// TIA Portal V20 export
// export: Created 2025-12-01T14:57:00.0403438Z, ExportSetting None, DisplayName Totally Integrated Automation Portal, DisplayVersion V20 Update 3, DisplayName TIA Portal Openness, DisplayVersion V20 Update 3, DisplayName TIA Portal Version Control Interface, DisplayVersion V20 Update 3, DisplayName STEP 7 Professional, DisplayVersion V20 Update 3, DisplayName STEP 7 Safety, DisplayVersion V20 Update 2, DisplayName WinCC Basic/Comfort/Advanced, DisplayVersion V20 Update 3, DisplayName WinCC Professional, DisplayVersion V20 Update 3, DisplayName WinCC Unified, DisplayVersion V20 Update 3
FUNCTION "FC427_TL_Sep_Salida_Bidi" : Void   // FC427, LAD
{ S7_Optimized_Access := 'FALSE' }
AUTHOR : TLigero
NAME : 20160208
VERSION : 3.1
// FECHA:    27/07/2014  AUTOR: G.Martin
// INSTALACION: Magyar Posta
// //////////////////////////////////
// // Registro Incidencias   ////////
// //////////////////////////////////
// FECHA:21/10/14   AUTOR MODIFICACION: N.Rodriguez
// DESCRIPCION: 
// Adaptación de la función al estandar actual
// 
// FECHA:   AUTOR MODIFICACION: 
// DESCRIPCION:
// stored: AutoNumber false, SetENOAutomatically false
   VAR_INPUT
      Mesa : UInt;
      En_Tension : Bool;
      Phs_Tx_E1 : Bool;   // Se utiliza esta fotocelula en caga E1-E3
      Phs_Tx_E3 : Bool;   // Se utiliza esta fotocelula en caga E3-E1
      Termico_Tx : Bool;
      Avance_E1_Tx_Ok : Bool;   // Avance con dirección E1-E3
      Avance_E3_Tx_Ok : Bool;   // Avance con dirección E3-E1
      Modo_Pasoapaso_Tx : Bool;
      Direccion_Inv_Tx : Bool;
      AVTF_Ent_M1 : Bool;
      AVTF_Ent_M3 : Bool;
      PTF_Sal_M1 : Bool;
      NXT_Avance_M1 : Bool;
      PTF_Sal_M3 : Bool;
      NXT_Avance_M3 : Bool;
      V_Ausencia_Tms : UDInt;
      V_Paro : UDInt;
      V_Separacion : UDInt;
      V_Caja_Max : UDInt;
      V_TOut_Tx_Mx : UDInt;
      V_Acumulacion : UDInt;
      V_Ausencia : UDInt;
   END_VAR
   VAR_OUTPUT
      PTF_Ent_M1 : Bool;
      PTF_Ent_M3 : Bool;
      AVTF_Sal_M1 : Bool;
      AVTF_Sal_M3 : Bool;
   END_VAR
   VAR_IN_OUT
      NXT_Descarga_Act_M1 : Bool;
      NXT_Descarga_Act_M3 : Bool;
      Carga_Activa_Tx : Bool;
      Carga_Activa_Inv_TX : Bool;
      MAUX_FN_Avtf : Bool;
      MAUX_FN_Direc : Bool;
      MAUX_FP_Direc : Bool;
      Mem_CNT_Tmp_AUS : Bool;
      Mem_CNT_Tmp_Paro_Tx : Bool;
      Mem_CNT_Acumulacion : Bool;
   END_VAR
   VAR_TEMP
      CNT_Sep : Word;
      CNT_Sep_FORZ_Sep : Int;
      Aux_Parar : Bool;
      Mem_CNT_Separacion : Bool;
      mem_atasco : Bool;
      fp_direc : Bool;
      fn_direc : Bool;
      mem_atasco_inv : Bool;
      ok_tension : Bool;
   END_VAR
   VAR_TEMP   // added for the SCL form of the ladder/FBD networks
      _w1 : Bool;
      _w2 : Bool;
   END_VAR
BEGIN

REGION Network 1: Marca General Error
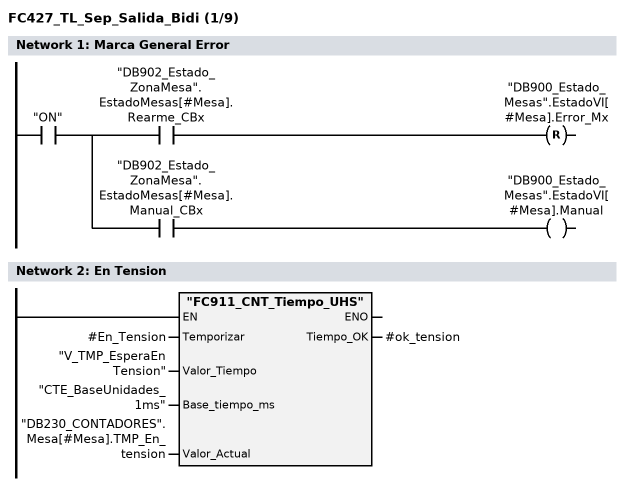
   RUNG wire#powerrail
      Contact( "ON" )
      wire#w1
      Contact( "DB902_Estado_ZonaMesa".EstadoMesas[#Mesa].Rearme_CBx )
      R_Coil( "DB900_Estado_Mesas".EstadoVI[#Mesa].Error_Mx )
   END_RUNG
   RUNG wire#w1
      Contact( "DB902_Estado_ZonaMesa".EstadoMesas[#Mesa].Manual_CBx )
      Coil( "DB900_Estado_Mesas".EstadoVI[#Mesa].Manual )
   END_RUNG
   // the same network as SCL:
   IF "ON" AND "DB902_Estado_ZonaMesa".EstadoMesas[#Mesa].Rearme_CBx THEN
       "DB900_Estado_Mesas".EstadoVI[#Mesa].Error_Mx := FALSE;
   END_IF;
   "DB900_Estado_Mesas".EstadoVI[#Mesa].Manual := "ON" AND "DB902_Estado_ZonaMesa".EstadoMesas[#Mesa].Manual_CBx;
END_REGION

REGION Network 2: En Tension
   RUNG wire#powerrail
      "FC911_CNT_Tiempo_UHS"(Temporizar := #En_Tension, Valor_Tiempo := "V_TMP_EsperaEnTension", Base_tiempo_ms := "CTE_BaseUnidades_1ms", Valor_Actual := "DB230_CONTADORES".Mesa[#Mesa].TMP_En_tension, Tiempo_OK => #ok_tension)
   END_RUNG
   // the same network as SCL:
   "FC911_CNT_Tiempo_UHS"(Temporizar := #En_Tension,
                          Valor_Tiempo := "V_TMP_EsperaEnTension",
                          Base_tiempo_ms := "CTE_BaseUnidades_1ms",
                          Valor_Actual := "DB230_CONTADORES".Mesa[#Mesa].TMP_En_tension,
                          Tiempo_OK => #ok_tension);
END_REGION

REGION Network 3: Reseteamos las marcas cuando hay cambio de direccion
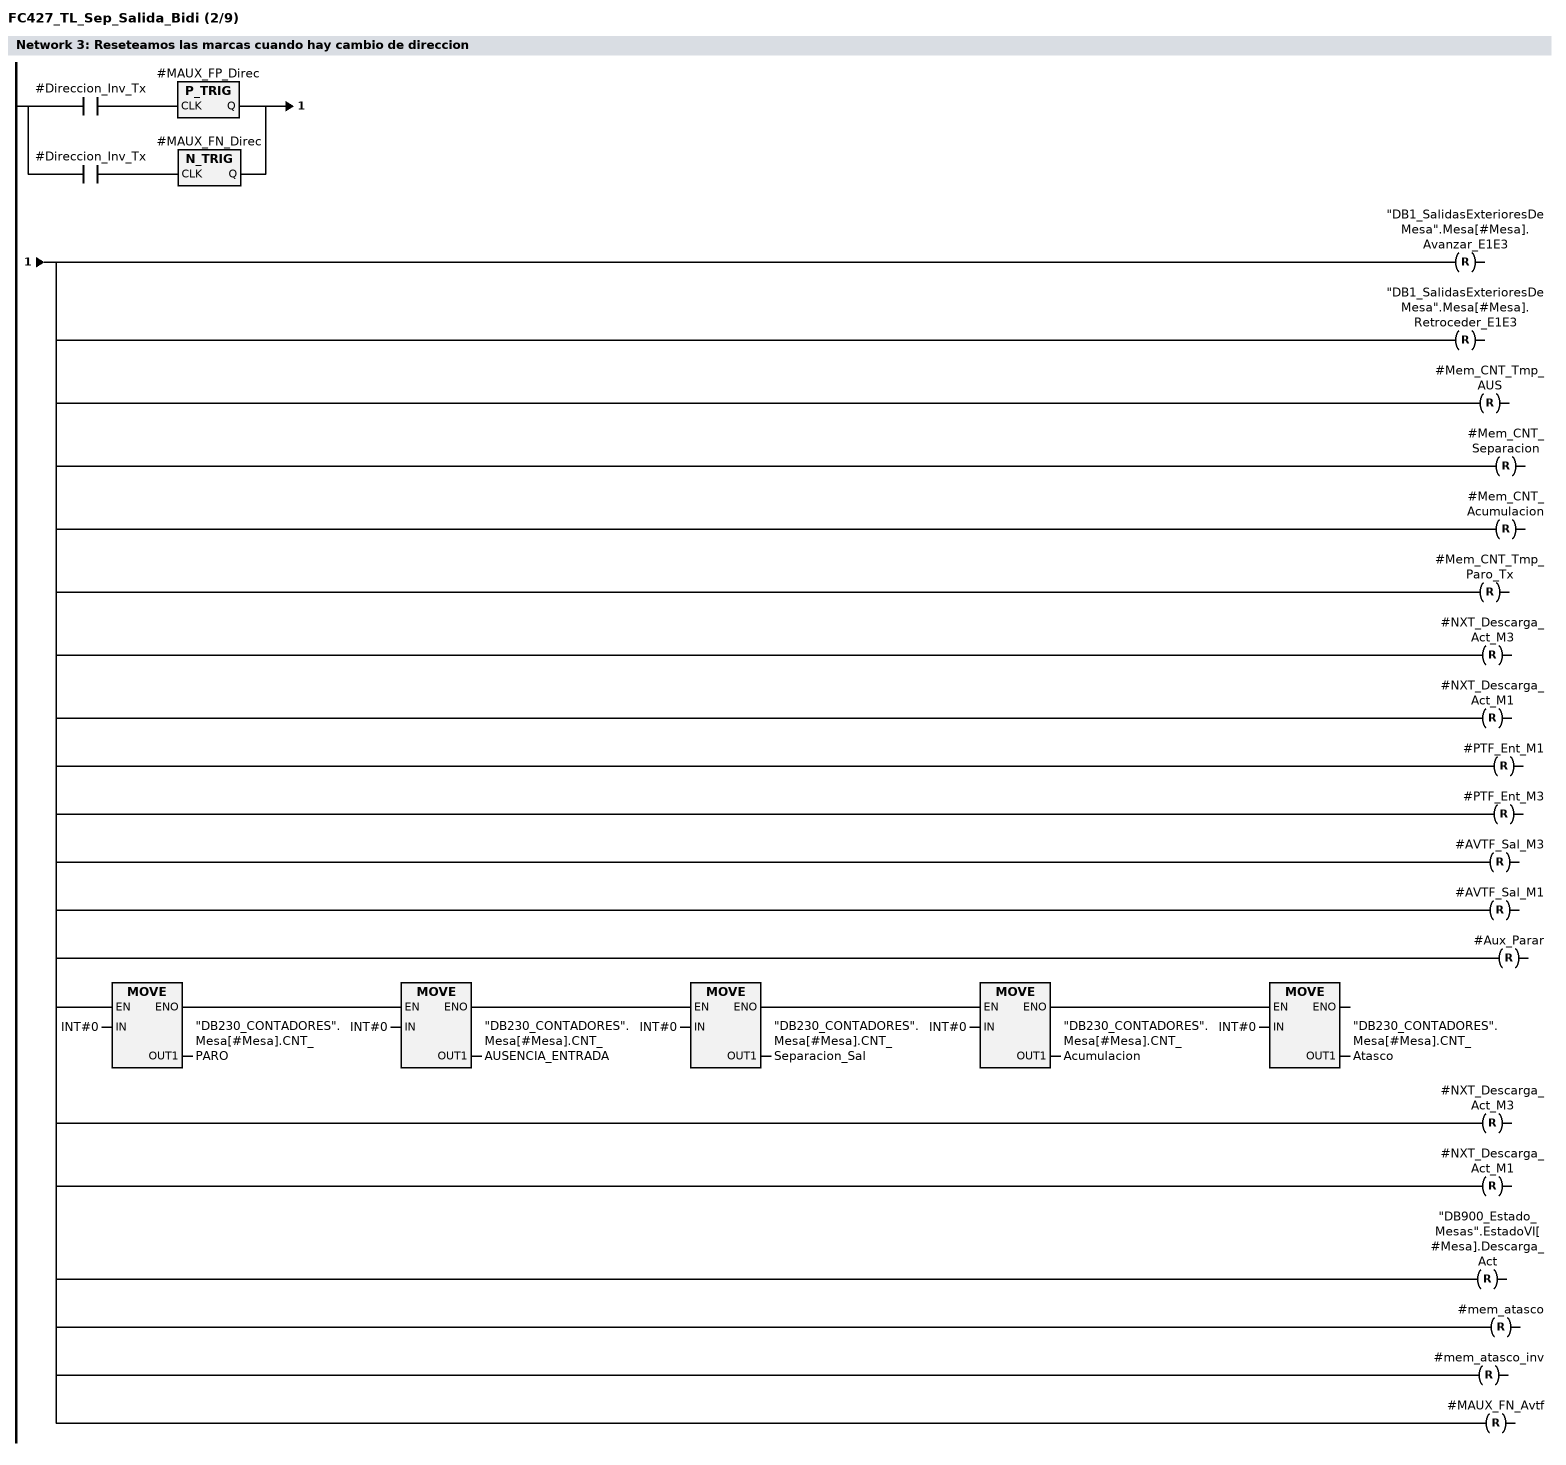
   RUNG wire#powerrail
      Contact( #Direccion_Inv_Tx )
      P_Trig( #MAUX_FP_Direc )
      wire#w1
      R_Coil( "DB1_SalidasExterioresDeMesa".Mesa[#Mesa].Avanzar_E1E3 )
   END_RUNG
   RUNG wire#powerrail
      Contact( #Direccion_Inv_Tx )
      N_Trig( #MAUX_FN_Direc )
   END_RUNG wire#w1
   RUNG wire#w1
      R_Coil( "DB1_SalidasExterioresDeMesa".Mesa[#Mesa].Retroceder_E1E3 )
   END_RUNG
   RUNG wire#w1
      R_Coil( #Mem_CNT_Tmp_AUS )
   END_RUNG
   RUNG wire#w1
      R_Coil( #Mem_CNT_Separacion )
   END_RUNG
   RUNG wire#w1
      R_Coil( #Mem_CNT_Acumulacion )
   END_RUNG
   RUNG wire#w1
      R_Coil( #Mem_CNT_Tmp_Paro_Tx )
   END_RUNG
   RUNG wire#w1
      R_Coil( #NXT_Descarga_Act_M3 )
   END_RUNG
   RUNG wire#w1
      R_Coil( #NXT_Descarga_Act_M1 )
   END_RUNG
   RUNG wire#w1
      R_Coil( #PTF_Ent_M1 )
   END_RUNG
   RUNG wire#w1
      R_Coil( #PTF_Ent_M3 )
   END_RUNG
   RUNG wire#w1
      R_Coil( #AVTF_Sal_M3 )
   END_RUNG
   RUNG wire#w1
      R_Coil( #AVTF_Sal_M1 )
   END_RUNG
   RUNG wire#w1
      R_Coil( #Aux_Parar )
   END_RUNG
   RUNG wire#w1
      { S7_GenerateENO := "TRUE" } Move(in := INT#0, out1 => "DB230_CONTADORES".Mesa[#Mesa].CNT_PARO)
      { S7_GenerateENO := "TRUE" } Move(in := INT#0, out1 => "DB230_CONTADORES".Mesa[#Mesa].CNT_AUSENCIA_ENTRADA)
      { S7_GenerateENO := "TRUE" } Move(in := INT#0, out1 => "DB230_CONTADORES".Mesa[#Mesa].CNT_Separacion_Sal)
      { S7_GenerateENO := "TRUE" } Move(in := INT#0, out1 => "DB230_CONTADORES".Mesa[#Mesa].CNT_Acumulacion)
      { S7_GenerateENO := "TRUE" } Move(in := INT#0, out1 => "DB230_CONTADORES".Mesa[#Mesa].CNT_Atasco)
   END_RUNG
   RUNG wire#w1
      R_Coil( #NXT_Descarga_Act_M3 )
   END_RUNG
   RUNG wire#w1
      R_Coil( #NXT_Descarga_Act_M1 )
   END_RUNG
   RUNG wire#w1
      R_Coil( "DB900_Estado_Mesas".EstadoVI[#Mesa].Descarga_Act )
   END_RUNG
   RUNG wire#w1
      R_Coil( #mem_atasco )
   END_RUNG
   RUNG wire#w1
      R_Coil( #mem_atasco_inv )
   END_RUNG
   RUNG wire#w1
      R_Coil( #MAUX_FN_Avtf )
   END_RUNG
   // the same network as SCL:
   // ENO of a box is taken as its EN; it also drops when the box reports an error
   #_w1 := #Direccion_Inv_Tx AND NOT #MAUX_FP_Direc;   // rising edge
   #MAUX_FP_Direc := #Direccion_Inv_Tx;
   #_w2 := NOT #Direccion_Inv_Tx AND #MAUX_FN_Direc;   // falling edge
   #MAUX_FN_Direc := #Direccion_Inv_Tx;
   IF #_w1 OR #_w2 THEN
       "DB1_SalidasExterioresDeMesa".Mesa[#Mesa].Avanzar_E1E3 := FALSE;
       "DB1_SalidasExterioresDeMesa".Mesa[#Mesa].Retroceder_E1E3 := FALSE;
       #Mem_CNT_Tmp_AUS := FALSE;
       #Mem_CNT_Separacion := FALSE;
       #Mem_CNT_Acumulacion := FALSE;
       #Mem_CNT_Tmp_Paro_Tx := FALSE;
       #NXT_Descarga_Act_M3 := FALSE;
       #NXT_Descarga_Act_M1 := FALSE;
       #PTF_Ent_M1 := FALSE;
       #PTF_Ent_M3 := FALSE;
       #AVTF_Sal_M3 := FALSE;
       #AVTF_Sal_M1 := FALSE;
       #Aux_Parar := FALSE;
       "DB230_CONTADORES".Mesa[#Mesa].CNT_PARO := INT#0;
       "DB230_CONTADORES".Mesa[#Mesa].CNT_AUSENCIA_ENTRADA := INT#0;
       "DB230_CONTADORES".Mesa[#Mesa].CNT_Separacion_Sal := INT#0;
       "DB230_CONTADORES".Mesa[#Mesa].CNT_Acumulacion := INT#0;
       "DB230_CONTADORES".Mesa[#Mesa].CNT_Atasco := INT#0;
       #NXT_Descarga_Act_M3 := FALSE;
       #NXT_Descarga_Act_M1 := FALSE;
       "DB900_Estado_Mesas".EstadoVI[#Mesa].Descarga_Act := FALSE;
       #mem_atasco := FALSE;
       #mem_atasco_inv := FALSE;
       #MAUX_FN_Avtf := FALSE;
   END_IF;
END_REGION

REGION Network 4: #Direccion_Inv_Tx
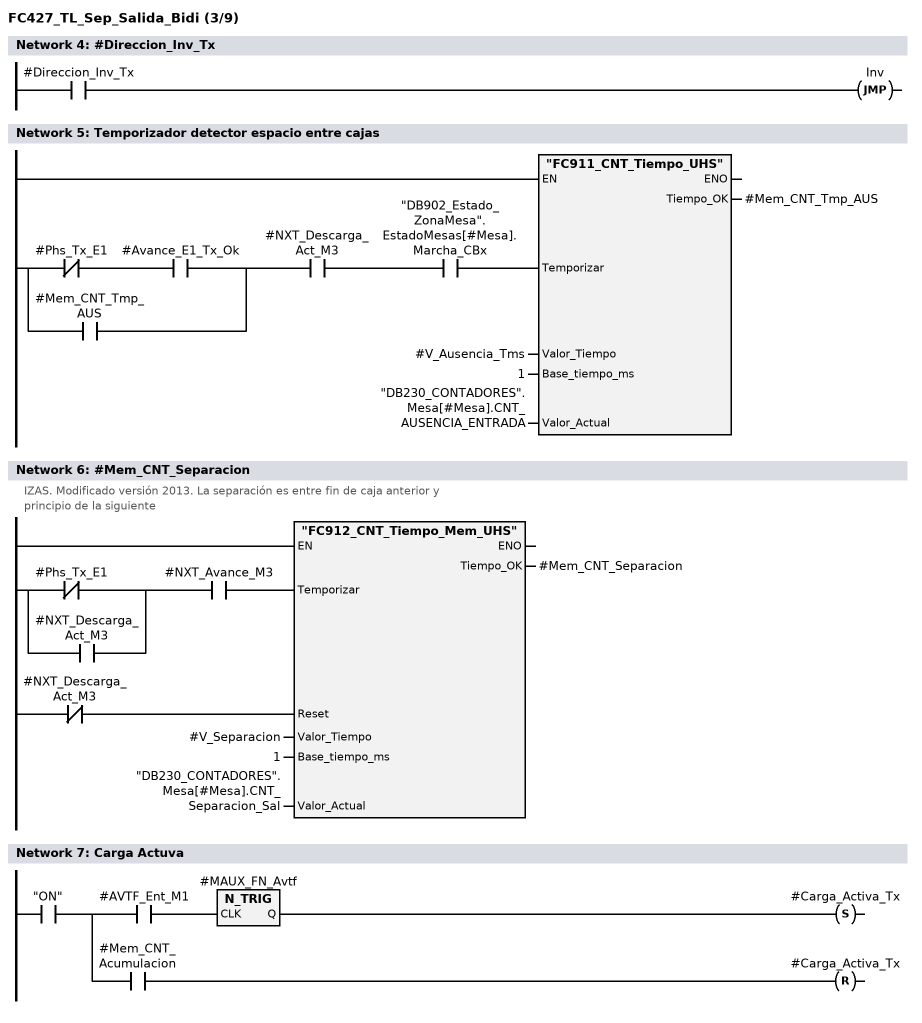
   RUNG wire#powerrail
      Contact( #Direccion_Inv_Tx )
      JumpCoil( Inv )
   END_RUNG
   // the same network as SCL:
   IF #Direccion_Inv_Tx THEN GOTO Inv; END_IF;
END_REGION

REGION Network 5: Temporizador detector espacio entre cajas
   RUNG wire#powerrail
      "FC911_CNT_Tiempo_UHS"(Temporizar := wire#w2, Valor_Tiempo := #V_Ausencia_Tms, Base_tiempo_ms := 1, Valor_Actual := "DB230_CONTADORES".Mesa[#Mesa].CNT_AUSENCIA_ENTRADA, Tiempo_OK => #Mem_CNT_Tmp_AUS)
   END_RUNG
   RUNG wire#powerrail
      I_Contact( #Phs_Tx_E1 )
      Contact( #Avance_E1_Tx_Ok )
      wire#w1
      Contact( #NXT_Descarga_Act_M3 )
      Contact( "DB902_Estado_ZonaMesa".EstadoMesas[#Mesa].Marcha_CBx )
   END_RUNG wire#w2
   RUNG wire#powerrail
      Contact( #Mem_CNT_Tmp_AUS )
   END_RUNG wire#w1
   // the same network as SCL:
   "FC911_CNT_Tiempo_UHS"(Temporizar := ((NOT #Phs_Tx_E1 AND #Avance_E1_Tx_Ok) OR #Mem_CNT_Tmp_AUS) AND #NXT_Descarga_Act_M3 AND "DB902_Estado_ZonaMesa".EstadoMesas[#Mesa].Marcha_CBx,
                          Valor_Tiempo := #V_Ausencia_Tms,
                          Base_tiempo_ms := 1,
                          Valor_Actual := "DB230_CONTADORES".Mesa[#Mesa].CNT_AUSENCIA_ENTRADA,
                          Tiempo_OK => #Mem_CNT_Tmp_AUS);
END_REGION

REGION Network 6: #Mem_CNT_Separacion
   // IZAS. Modificado versión 2013. La separación es entre fin de caja anterior y 
   // principio de la siguiente
   RUNG wire#powerrail
      "FC912_CNT_Tiempo_Mem_UHS"(Temporizar := wire#w2, Reset := wire#w3, Valor_Tiempo := #V_Separacion, Base_tiempo_ms := 1, Valor_Actual := "DB230_CONTADORES".Mesa[#Mesa].CNT_Separacion_Sal, Tiempo_OK => #Mem_CNT_Separacion)
   END_RUNG
   RUNG wire#powerrail
      I_Contact( #Phs_Tx_E1 )
      wire#w1
      Contact( #NXT_Avance_M3 )
   END_RUNG wire#w2
   RUNG wire#powerrail
      Contact( #NXT_Descarga_Act_M3 )
   END_RUNG wire#w1
   RUNG wire#powerrail
      I_Contact( #NXT_Descarga_Act_M3 )
   END_RUNG wire#w3
   // the same network as SCL:
   "FC912_CNT_Tiempo_Mem_UHS"(Temporizar := (NOT #Phs_Tx_E1 OR #NXT_Descarga_Act_M3) AND #NXT_Avance_M3,
                           Reset := NOT #NXT_Descarga_Act_M3,
                           Valor_Tiempo := #V_Separacion,
                           Base_tiempo_ms := 1,
                           Valor_Actual := "DB230_CONTADORES".Mesa[#Mesa].CNT_Separacion_Sal,
                           Tiempo_OK => #Mem_CNT_Separacion);
END_REGION

REGION Network 7: Carga Actuva
   RUNG wire#powerrail
      Contact( "ON" )
      wire#w1
      Contact( #AVTF_Ent_M1 )
      N_Trig( #MAUX_FN_Avtf )
      S_Coil( #Carga_Activa_Tx )
   END_RUNG
   RUNG wire#w1
      Contact( #Mem_CNT_Acumulacion )
      R_Coil( #Carga_Activa_Tx )
   END_RUNG
   // the same network as SCL:
   #_w1 := "ON" AND #AVTF_Ent_M1;
   #_w2 := NOT #_w1 AND #MAUX_FN_Avtf;   // falling edge
   #MAUX_FN_Avtf := #_w1;
   IF #_w2 THEN #Carga_Activa_Tx := TRUE; END_IF;
   IF "ON" AND #Mem_CNT_Acumulacion THEN #Carga_Activa_Tx := FALSE; END_IF;
END_REGION

REGION Network 8: Mem_CNT_Acumulacion
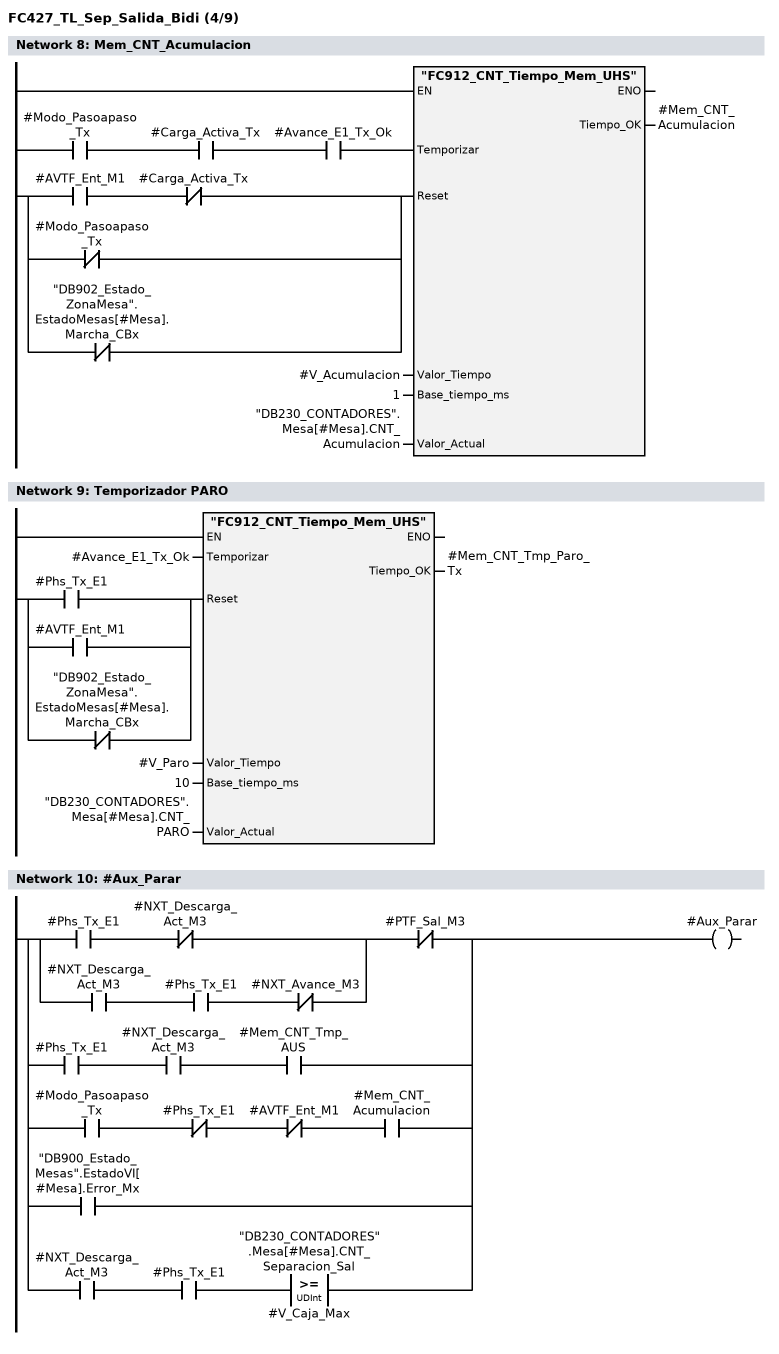
   RUNG wire#powerrail
      "FC912_CNT_Tiempo_Mem_UHS"(Temporizar := wire#w1, Reset := wire#w2, Valor_Tiempo := #V_Acumulacion, Base_tiempo_ms := 1, Valor_Actual := "DB230_CONTADORES".Mesa[#Mesa].CNT_Acumulacion, Tiempo_OK => #Mem_CNT_Acumulacion)
   END_RUNG
   RUNG wire#powerrail
      Contact( #Modo_Pasoapaso_Tx )
      Contact( #Carga_Activa_Tx )
      Contact( #Avance_E1_Tx_Ok )
   END_RUNG wire#w1
   RUNG wire#powerrail
      Contact( #AVTF_Ent_M1 )
      I_Contact( #Carga_Activa_Tx )
   END_RUNG wire#w2
   RUNG wire#powerrail
      I_Contact( #Modo_Pasoapaso_Tx )
   END_RUNG wire#w2
   RUNG wire#powerrail
      I_Contact( "DB902_Estado_ZonaMesa".EstadoMesas[#Mesa].Marcha_CBx )
   END_RUNG wire#w2
   // the same network as SCL:
   "FC912_CNT_Tiempo_Mem_UHS"(Temporizar := #Modo_Pasoapaso_Tx AND #Carga_Activa_Tx AND #Avance_E1_Tx_Ok,
                           Reset := (#AVTF_Ent_M1 AND NOT #Carga_Activa_Tx) OR NOT #Modo_Pasoapaso_Tx OR NOT "DB902_Estado_ZonaMesa".EstadoMesas[#Mesa].Marcha_CBx,
                           Valor_Tiempo := #V_Acumulacion,
                           Base_tiempo_ms := 1,
                           Valor_Actual := "DB230_CONTADORES".Mesa[#Mesa].CNT_Acumulacion,
                           Tiempo_OK => #Mem_CNT_Acumulacion);
END_REGION

REGION Network 9: Temporizador PARO
   RUNG wire#powerrail
      "FC912_CNT_Tiempo_Mem_UHS"(Reset := wire#w1, Temporizar := #Avance_E1_Tx_Ok, Valor_Tiempo := #V_Paro, Base_tiempo_ms := 10, Valor_Actual := "DB230_CONTADORES".Mesa[#Mesa].CNT_PARO, Tiempo_OK => #Mem_CNT_Tmp_Paro_Tx)
   END_RUNG
   RUNG wire#powerrail
      Contact( #Phs_Tx_E1 )
   END_RUNG wire#w1
   RUNG wire#powerrail
      Contact( #AVTF_Ent_M1 )
   END_RUNG wire#w1
   RUNG wire#powerrail
      I_Contact( "DB902_Estado_ZonaMesa".EstadoMesas[#Mesa].Marcha_CBx )
   END_RUNG wire#w1
   // the same network as SCL:
   "FC912_CNT_Tiempo_Mem_UHS"(Temporizar := #Avance_E1_Tx_Ok,
                           Reset := #Phs_Tx_E1 OR #AVTF_Ent_M1 OR NOT "DB902_Estado_ZonaMesa".EstadoMesas[#Mesa].Marcha_CBx,
                           Valor_Tiempo := #V_Paro,
                           Base_tiempo_ms := 10,
                           Valor_Actual := "DB230_CONTADORES".Mesa[#Mesa].CNT_PARO,
                           Tiempo_OK => #Mem_CNT_Tmp_Paro_Tx);
END_REGION

REGION Network 10: #Aux_Parar
   RUNG wire#powerrail
      Contact( #Phs_Tx_E1 )
      I_Contact( #NXT_Descarga_Act_M3 )
      wire#w1
      I_Contact( #PTF_Sal_M3 )
      wire#w2
      Coil( #Aux_Parar )
   END_RUNG
   RUNG wire#powerrail
      Contact( #NXT_Descarga_Act_M3 )
      Contact( #Phs_Tx_E1 )
      I_Contact( #NXT_Avance_M3 )
   END_RUNG wire#w1
   RUNG wire#powerrail
      Contact( #Phs_Tx_E1 )
      Contact( #NXT_Descarga_Act_M3 )
      Contact( #Mem_CNT_Tmp_AUS )
   END_RUNG wire#w2
   RUNG wire#powerrail
      Contact( #Modo_Pasoapaso_Tx )
      I_Contact( #Phs_Tx_E1 )
      I_Contact( #AVTF_Ent_M1 )
      Contact( #Mem_CNT_Acumulacion )
   END_RUNG wire#w2
   RUNG wire#powerrail
      Contact( "DB900_Estado_Mesas".EstadoVI[#Mesa].Error_Mx )
   END_RUNG wire#w2
   RUNG wire#powerrail
      Contact( #NXT_Descarga_Act_M3 )
      Contact( #Phs_Tx_E1 )
      { S7_Templates := "SrcType := UDInt" } GE_Contact(in1 := "DB230_CONTADORES".Mesa[#Mesa].CNT_Separacion_Sal, in2 := #V_Caja_Max)
   END_RUNG wire#w2
   // the same network as SCL:
   #Aux_Parar := (((#Phs_Tx_E1 AND NOT #NXT_Descarga_Act_M3) OR (#NXT_Descarga_Act_M3 AND #Phs_Tx_E1 AND NOT #NXT_Avance_M3)) AND NOT #PTF_Sal_M3) OR (#Phs_Tx_E1 AND #NXT_Descarga_Act_M3 AND #Mem_CNT_Tmp_AUS) OR (#Modo_Pasoapaso_Tx AND NOT #Phs_Tx_E1 AND NOT #AVTF_Ent_M1 AND #Mem_CNT_Acumulacion) OR "DB900_Estado_Mesas".EstadoVI[#Mesa].Error_Mx OR (#NXT_Descarga_Act_M3 AND #Phs_Tx_E1 AND ("DB230_CONTADORES".Mesa[#Mesa].CNT_Separacion_Sal >= #V_Caja_Max));
END_REGION

REGION Network 11: Memoria Transporte en descarga
   // modificado despues de hablar con carlos.
   // Antes el reseteo era con la variable del contador negada
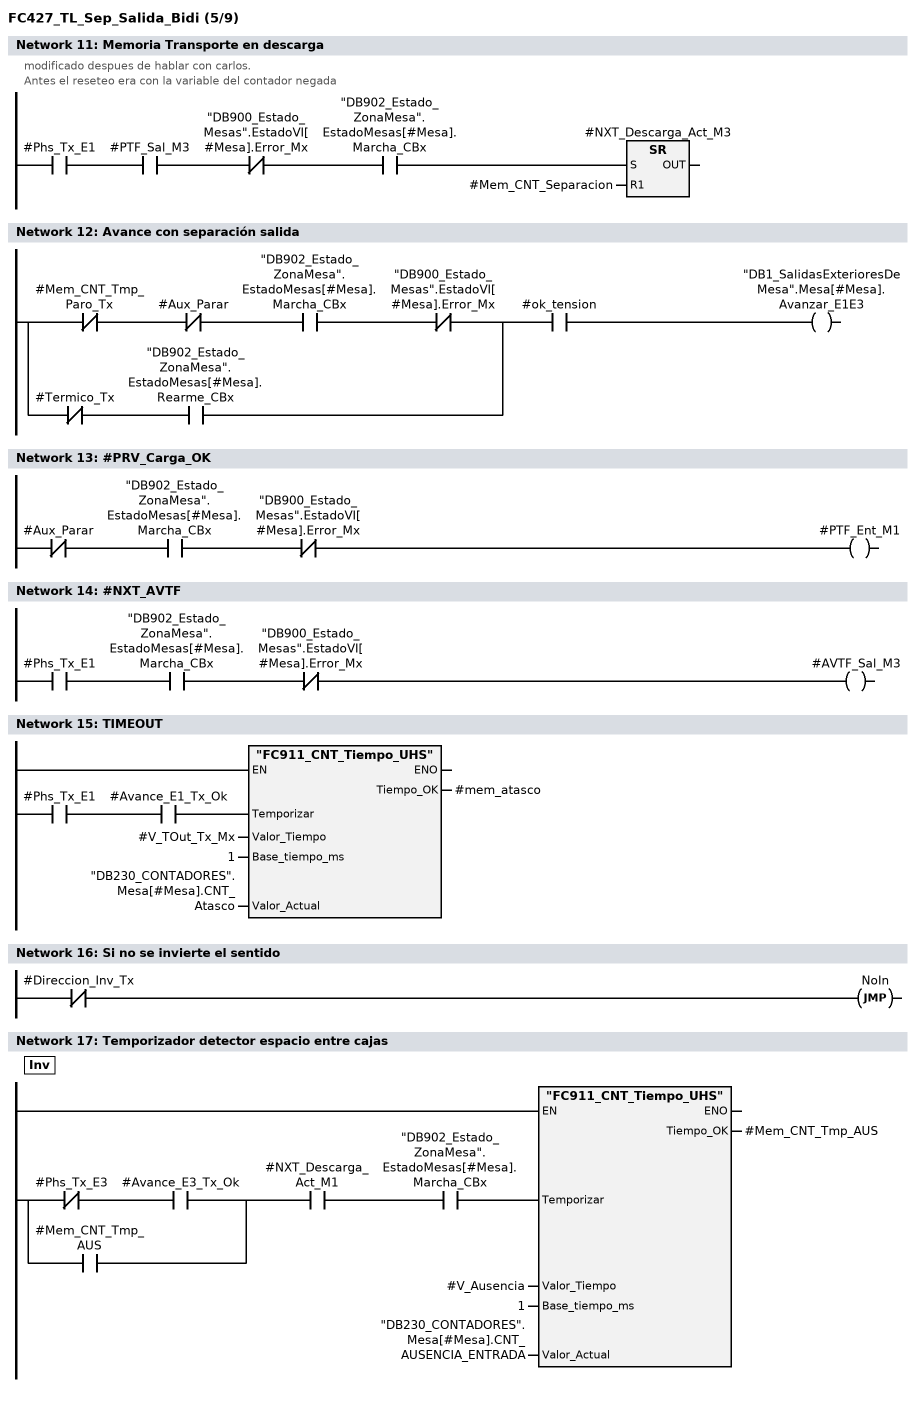
   RUNG wire#powerrail
      Contact( #Phs_Tx_E1 )
      Contact( #PTF_Sal_M3 )
      I_Contact( "DB900_Estado_Mesas".EstadoVI[#Mesa].Error_Mx )
      Contact( "DB902_Estado_ZonaMesa".EstadoMesas[#Mesa].Marcha_CBx )
      S_SR(operand := #NXT_Descarga_Act_M3, r1 := #Mem_CNT_Separacion)
   END_RUNG
   // the same network as SCL:
   IF #Phs_Tx_E1 AND #PTF_Sal_M3 AND NOT "DB900_Estado_Mesas".EstadoVI[#Mesa].Error_Mx AND "DB902_Estado_ZonaMesa".EstadoMesas[#Mesa].Marcha_CBx THEN
       #NXT_Descarga_Act_M3 := TRUE;   // SR flip-flop
   END_IF;
   IF #Mem_CNT_Separacion THEN #NXT_Descarga_Act_M3 := FALSE; END_IF;
END_REGION

REGION Network 12: Avance con separación salida
   RUNG wire#powerrail
      I_Contact( #Mem_CNT_Tmp_Paro_Tx )
      I_Contact( #Aux_Parar )
      Contact( "DB902_Estado_ZonaMesa".EstadoMesas[#Mesa].Marcha_CBx )
      I_Contact( "DB900_Estado_Mesas".EstadoVI[#Mesa].Error_Mx )
      wire#w1
      Contact( #ok_tension )
      Coil( "DB1_SalidasExterioresDeMesa".Mesa[#Mesa].Avanzar_E1E3 )
   END_RUNG
   RUNG wire#powerrail
      I_Contact( #Termico_Tx )
      Contact( "DB902_Estado_ZonaMesa".EstadoMesas[#Mesa].Rearme_CBx )
   END_RUNG wire#w1
   // the same network as SCL:
   "DB1_SalidasExterioresDeMesa".Mesa[#Mesa].Avanzar_E1E3 := ((NOT #Mem_CNT_Tmp_Paro_Tx AND NOT #Aux_Parar AND "DB902_Estado_ZonaMesa".EstadoMesas[#Mesa].Marcha_CBx AND NOT "DB900_Estado_Mesas".EstadoVI[#Mesa].Error_Mx) OR (NOT #Termico_Tx AND "DB902_Estado_ZonaMesa".EstadoMesas[#Mesa].Rearme_CBx)) AND #ok_tension;
END_REGION

REGION Network 13: #PRV_Carga_OK
   RUNG wire#powerrail
      I_Contact( #Aux_Parar )
      Contact( "DB902_Estado_ZonaMesa".EstadoMesas[#Mesa].Marcha_CBx )
      I_Contact( "DB900_Estado_Mesas".EstadoVI[#Mesa].Error_Mx )
      Coil( #PTF_Ent_M1 )
   END_RUNG
   // the same network as SCL:
   #PTF_Ent_M1 := NOT #Aux_Parar AND "DB902_Estado_ZonaMesa".EstadoMesas[#Mesa].Marcha_CBx AND NOT "DB900_Estado_Mesas".EstadoVI[#Mesa].Error_Mx;
END_REGION

REGION Network 14: #NXT_AVTF
   RUNG wire#powerrail
      Contact( #Phs_Tx_E1 )
      Contact( "DB902_Estado_ZonaMesa".EstadoMesas[#Mesa].Marcha_CBx )
      I_Contact( "DB900_Estado_Mesas".EstadoVI[#Mesa].Error_Mx )
      Coil( #AVTF_Sal_M3 )
   END_RUNG
   // the same network as SCL:
   #AVTF_Sal_M3 := #Phs_Tx_E1 AND "DB902_Estado_ZonaMesa".EstadoMesas[#Mesa].Marcha_CBx AND NOT "DB900_Estado_Mesas".EstadoVI[#Mesa].Error_Mx;
END_REGION

REGION Network 15: TIMEOUT
   RUNG wire#powerrail
      "FC911_CNT_Tiempo_UHS"(Temporizar := wire#w1, Valor_Tiempo := #V_TOut_Tx_Mx, Base_tiempo_ms := 1, Valor_Actual := "DB230_CONTADORES".Mesa[#Mesa].CNT_Atasco, Tiempo_OK => #mem_atasco)
   END_RUNG
   RUNG wire#powerrail
      Contact( #Phs_Tx_E1 )
      Contact( #Avance_E1_Tx_Ok )
   END_RUNG wire#w1
   // the same network as SCL:
   "FC911_CNT_Tiempo_UHS"(Temporizar := #Phs_Tx_E1 AND #Avance_E1_Tx_Ok,
                          Valor_Tiempo := #V_TOut_Tx_Mx,
                          Base_tiempo_ms := 1,
                          Valor_Actual := "DB230_CONTADORES".Mesa[#Mesa].CNT_Atasco,
                          Tiempo_OK => #mem_atasco);
END_REGION

REGION Network 16: Si no se invierte el sentido
   RUNG wire#powerrail
      I_Contact( #Direccion_Inv_Tx )
      JumpCoil( NoIn )
   END_RUNG
   // the same network as SCL:
   IF NOT #Direccion_Inv_Tx THEN GOTO NoIn; END_IF;
END_REGION

REGION Network 17: Temporizador detector espacio entre cajas
   Label( Inv )
   RUNG wire#powerrail
      "FC911_CNT_Tiempo_UHS"(Temporizar := wire#w2, Valor_Tiempo := #V_Ausencia, Base_tiempo_ms := 1, Valor_Actual := "DB230_CONTADORES".Mesa[#Mesa].CNT_AUSENCIA_ENTRADA, Tiempo_OK => #Mem_CNT_Tmp_AUS)
   END_RUNG
   RUNG wire#powerrail
      I_Contact( #Phs_Tx_E3 )
      Contact( #Avance_E3_Tx_Ok )
      wire#w1
      Contact( #NXT_Descarga_Act_M1 )
      Contact( "DB902_Estado_ZonaMesa".EstadoMesas[#Mesa].Marcha_CBx )
   END_RUNG wire#w2
   RUNG wire#powerrail
      Contact( #Mem_CNT_Tmp_AUS )
   END_RUNG wire#w1
   // the same network as SCL:
   Inv:
   "FC911_CNT_Tiempo_UHS"(Temporizar := ((NOT #Phs_Tx_E3 AND #Avance_E3_Tx_Ok) OR #Mem_CNT_Tmp_AUS) AND #NXT_Descarga_Act_M1 AND "DB902_Estado_ZonaMesa".EstadoMesas[#Mesa].Marcha_CBx,
                          Valor_Tiempo := #V_Ausencia,
                          Base_tiempo_ms := 1,
                          Valor_Actual := "DB230_CONTADORES".Mesa[#Mesa].CNT_AUSENCIA_ENTRADA,
                          Tiempo_OK => #Mem_CNT_Tmp_AUS);
END_REGION

REGION Network 18: #Mem_CNT_Separacion
   // IZAS. Modificado versión 2013. La separación es entre fin de caja anterior y 
   // principio de la siguiente
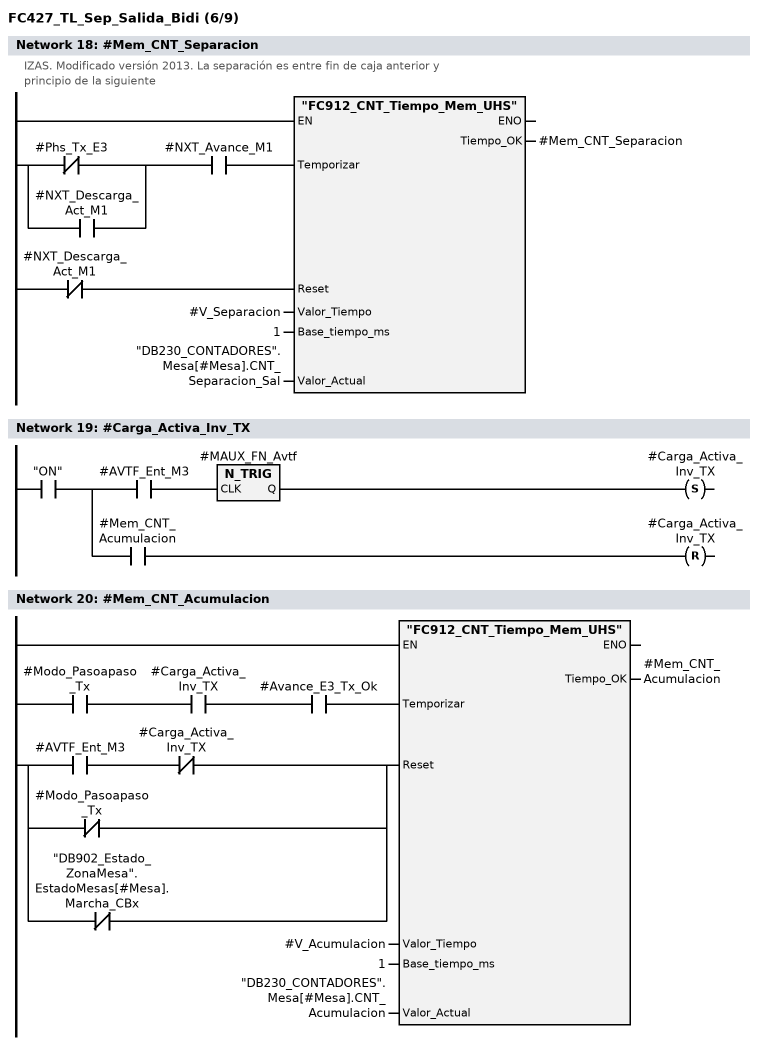
   RUNG wire#powerrail
      "FC912_CNT_Tiempo_Mem_UHS"(Temporizar := wire#w2, Reset := wire#w3, Valor_Tiempo := #V_Separacion, Base_tiempo_ms := 1, Valor_Actual := "DB230_CONTADORES".Mesa[#Mesa].CNT_Separacion_Sal, Tiempo_OK => #Mem_CNT_Separacion)
   END_RUNG
   RUNG wire#powerrail
      I_Contact( #Phs_Tx_E3 )
      wire#w1
      Contact( #NXT_Avance_M1 )
   END_RUNG wire#w2
   RUNG wire#powerrail
      Contact( #NXT_Descarga_Act_M1 )
   END_RUNG wire#w1
   RUNG wire#powerrail
      I_Contact( #NXT_Descarga_Act_M1 )
   END_RUNG wire#w3
   // the same network as SCL:
   "FC912_CNT_Tiempo_Mem_UHS"(Temporizar := (NOT #Phs_Tx_E3 OR #NXT_Descarga_Act_M1) AND #NXT_Avance_M1,
                           Reset := NOT #NXT_Descarga_Act_M1,
                           Valor_Tiempo := #V_Separacion,
                           Base_tiempo_ms := 1,
                           Valor_Actual := "DB230_CONTADORES".Mesa[#Mesa].CNT_Separacion_Sal,
                           Tiempo_OK => #Mem_CNT_Separacion);
END_REGION

REGION Network 19: #Carga_Activa_Inv_TX
   RUNG wire#powerrail
      Contact( "ON" )
      wire#w1
      Contact( #AVTF_Ent_M3 )
      N_Trig( #MAUX_FN_Avtf )
      S_Coil( #Carga_Activa_Inv_TX )
   END_RUNG
   RUNG wire#w1
      Contact( #Mem_CNT_Acumulacion )
      R_Coil( #Carga_Activa_Inv_TX )
   END_RUNG
   // the same network as SCL:
   #_w1 := "ON" AND #AVTF_Ent_M3;
   #_w2 := NOT #_w1 AND #MAUX_FN_Avtf;   // falling edge
   #MAUX_FN_Avtf := #_w1;
   IF #_w2 THEN #Carga_Activa_Inv_TX := TRUE; END_IF;
   IF "ON" AND #Mem_CNT_Acumulacion THEN #Carga_Activa_Inv_TX := FALSE; END_IF;
END_REGION

REGION Network 20: #Mem_CNT_Acumulacion
   RUNG wire#powerrail
      "FC912_CNT_Tiempo_Mem_UHS"(Temporizar := wire#w1, Reset := wire#w2, Valor_Tiempo := #V_Acumulacion, Base_tiempo_ms := 1, Valor_Actual := "DB230_CONTADORES".Mesa[#Mesa].CNT_Acumulacion, Tiempo_OK => #Mem_CNT_Acumulacion)
   END_RUNG
   RUNG wire#powerrail
      Contact( #Modo_Pasoapaso_Tx )
      Contact( #Carga_Activa_Inv_TX )
      Contact( #Avance_E3_Tx_Ok )
   END_RUNG wire#w1
   RUNG wire#powerrail
      Contact( #AVTF_Ent_M3 )
      I_Contact( #Carga_Activa_Inv_TX )
   END_RUNG wire#w2
   RUNG wire#powerrail
      I_Contact( #Modo_Pasoapaso_Tx )
   END_RUNG wire#w2
   RUNG wire#powerrail
      I_Contact( "DB902_Estado_ZonaMesa".EstadoMesas[#Mesa].Marcha_CBx )
   END_RUNG wire#w2
   // the same network as SCL:
   "FC912_CNT_Tiempo_Mem_UHS"(Temporizar := #Modo_Pasoapaso_Tx AND #Carga_Activa_Inv_TX AND #Avance_E3_Tx_Ok,
                           Reset := (#AVTF_Ent_M3 AND NOT #Carga_Activa_Inv_TX) OR NOT #Modo_Pasoapaso_Tx OR NOT "DB902_Estado_ZonaMesa".EstadoMesas[#Mesa].Marcha_CBx,
                           Valor_Tiempo := #V_Acumulacion,
                           Base_tiempo_ms := 1,
                           Valor_Actual := "DB230_CONTADORES".Mesa[#Mesa].CNT_Acumulacion,
                           Tiempo_OK => #Mem_CNT_Acumulacion);
END_REGION

REGION Network 21: Temporizador PARO
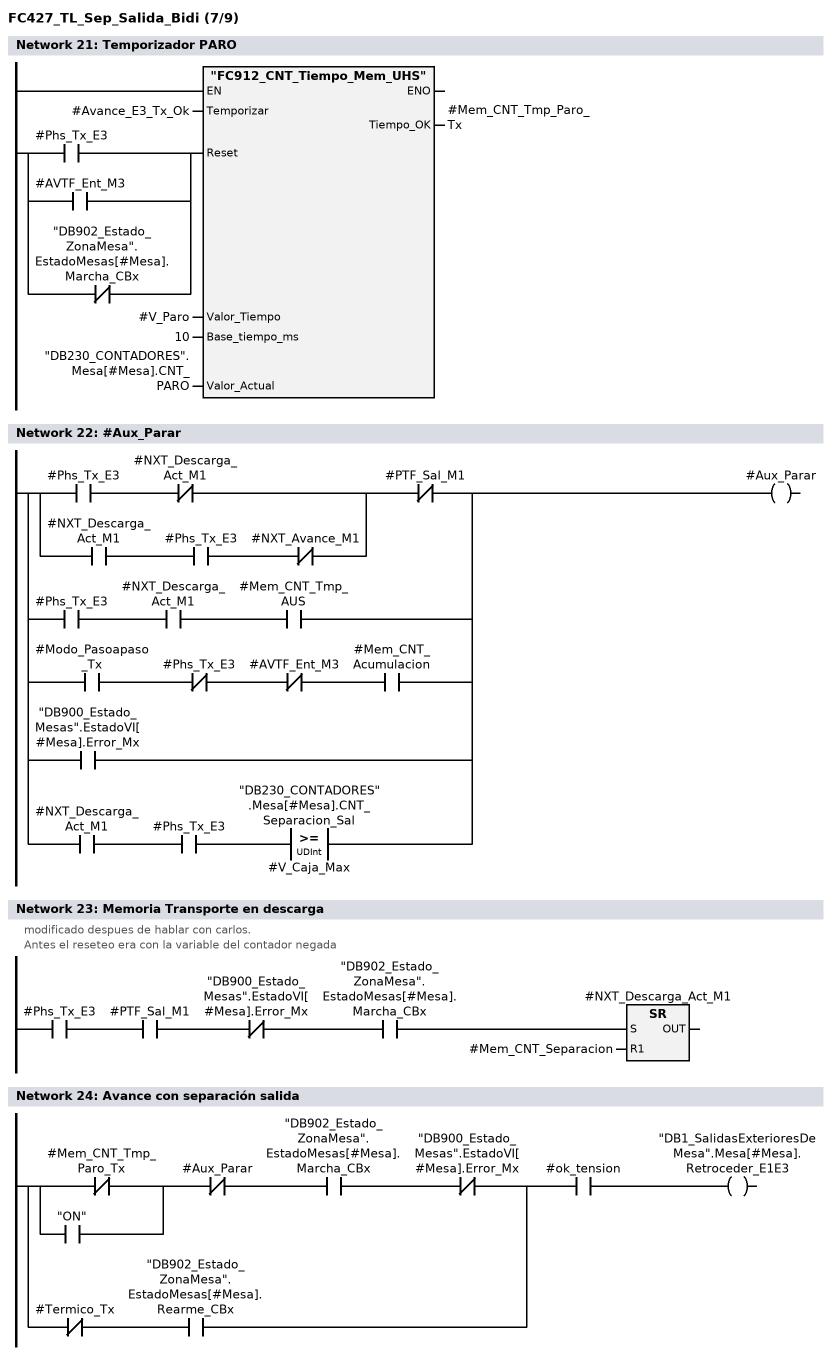
   RUNG wire#powerrail
      "FC912_CNT_Tiempo_Mem_UHS"(Reset := wire#w1, Temporizar := #Avance_E3_Tx_Ok, Valor_Tiempo := #V_Paro, Base_tiempo_ms := 10, Valor_Actual := "DB230_CONTADORES".Mesa[#Mesa].CNT_PARO, Tiempo_OK => #Mem_CNT_Tmp_Paro_Tx)
   END_RUNG
   RUNG wire#powerrail
      Contact( #Phs_Tx_E3 )
   END_RUNG wire#w1
   RUNG wire#powerrail
      Contact( #AVTF_Ent_M3 )
   END_RUNG wire#w1
   RUNG wire#powerrail
      I_Contact( "DB902_Estado_ZonaMesa".EstadoMesas[#Mesa].Marcha_CBx )
   END_RUNG wire#w1
   // the same network as SCL:
   "FC912_CNT_Tiempo_Mem_UHS"(Temporizar := #Avance_E3_Tx_Ok,
                           Reset := #Phs_Tx_E3 OR #AVTF_Ent_M3 OR NOT "DB902_Estado_ZonaMesa".EstadoMesas[#Mesa].Marcha_CBx,
                           Valor_Tiempo := #V_Paro,
                           Base_tiempo_ms := 10,
                           Valor_Actual := "DB230_CONTADORES".Mesa[#Mesa].CNT_PARO,
                           Tiempo_OK => #Mem_CNT_Tmp_Paro_Tx);
END_REGION

REGION Network 22: #Aux_Parar
   RUNG wire#powerrail
      Contact( #Phs_Tx_E3 )
      I_Contact( #NXT_Descarga_Act_M1 )
      wire#w1
      I_Contact( #PTF_Sal_M1 )
      wire#w2
      Coil( #Aux_Parar )
   END_RUNG
   RUNG wire#powerrail
      Contact( #NXT_Descarga_Act_M1 )
      Contact( #Phs_Tx_E3 )
      I_Contact( #NXT_Avance_M1 )
   END_RUNG wire#w1
   RUNG wire#powerrail
      Contact( #Phs_Tx_E3 )
      Contact( #NXT_Descarga_Act_M1 )
      Contact( #Mem_CNT_Tmp_AUS )
   END_RUNG wire#w2
   RUNG wire#powerrail
      Contact( #Modo_Pasoapaso_Tx )
      I_Contact( #Phs_Tx_E3 )
      I_Contact( #AVTF_Ent_M3 )
      Contact( #Mem_CNT_Acumulacion )
   END_RUNG wire#w2
   RUNG wire#powerrail
      Contact( "DB900_Estado_Mesas".EstadoVI[#Mesa].Error_Mx )
   END_RUNG wire#w2
   RUNG wire#powerrail
      Contact( #NXT_Descarga_Act_M1 )
      Contact( #Phs_Tx_E3 )
      { S7_Templates := "SrcType := UDInt" } GE_Contact(in1 := "DB230_CONTADORES".Mesa[#Mesa].CNT_Separacion_Sal, in2 := #V_Caja_Max)
   END_RUNG wire#w2
   // the same network as SCL:
   #Aux_Parar := (((#Phs_Tx_E3 AND NOT #NXT_Descarga_Act_M1) OR (#NXT_Descarga_Act_M1 AND #Phs_Tx_E3 AND NOT #NXT_Avance_M1)) AND NOT #PTF_Sal_M1) OR (#Phs_Tx_E3 AND #NXT_Descarga_Act_M1 AND #Mem_CNT_Tmp_AUS) OR (#Modo_Pasoapaso_Tx AND NOT #Phs_Tx_E3 AND NOT #AVTF_Ent_M3 AND #Mem_CNT_Acumulacion) OR "DB900_Estado_Mesas".EstadoVI[#Mesa].Error_Mx OR (#NXT_Descarga_Act_M1 AND #Phs_Tx_E3 AND ("DB230_CONTADORES".Mesa[#Mesa].CNT_Separacion_Sal >= #V_Caja_Max));
END_REGION

REGION Network 23: Memoria Transporte en descarga
   // modificado despues de hablar con carlos.
   // Antes el reseteo era con la variable del contador negada
   RUNG wire#powerrail
      Contact( #Phs_Tx_E3 )
      Contact( #PTF_Sal_M1 )
      I_Contact( "DB900_Estado_Mesas".EstadoVI[#Mesa].Error_Mx )
      Contact( "DB902_Estado_ZonaMesa".EstadoMesas[#Mesa].Marcha_CBx )
      S_SR(operand := #NXT_Descarga_Act_M1, r1 := #Mem_CNT_Separacion)
   END_RUNG
   // the same network as SCL:
   IF #Phs_Tx_E3 AND #PTF_Sal_M1 AND NOT "DB900_Estado_Mesas".EstadoVI[#Mesa].Error_Mx AND "DB902_Estado_ZonaMesa".EstadoMesas[#Mesa].Marcha_CBx THEN
       #NXT_Descarga_Act_M1 := TRUE;   // SR flip-flop
   END_IF;
   IF #Mem_CNT_Separacion THEN #NXT_Descarga_Act_M1 := FALSE; END_IF;
END_REGION

REGION Network 24: Avance con separación salida
   RUNG wire#powerrail
      I_Contact( #Mem_CNT_Tmp_Paro_Tx )
      wire#w1
      I_Contact( #Aux_Parar )
      Contact( "DB902_Estado_ZonaMesa".EstadoMesas[#Mesa].Marcha_CBx )
      I_Contact( "DB900_Estado_Mesas".EstadoVI[#Mesa].Error_Mx )
      wire#w2
      Contact( #ok_tension )
      Coil( "DB1_SalidasExterioresDeMesa".Mesa[#Mesa].Retroceder_E1E3 )
   END_RUNG
   RUNG wire#powerrail
      Contact( "ON" )
   END_RUNG wire#w1
   RUNG wire#powerrail
      I_Contact( #Termico_Tx )
      Contact( "DB902_Estado_ZonaMesa".EstadoMesas[#Mesa].Rearme_CBx )
   END_RUNG wire#w2
   // the same network as SCL:
   "DB1_SalidasExterioresDeMesa".Mesa[#Mesa].Retroceder_E1E3 := (((NOT #Mem_CNT_Tmp_Paro_Tx OR "ON") AND NOT #Aux_Parar AND "DB902_Estado_ZonaMesa".EstadoMesas[#Mesa].Marcha_CBx AND NOT "DB900_Estado_Mesas".EstadoVI[#Mesa].Error_Mx) OR (NOT #Termico_Tx AND "DB902_Estado_ZonaMesa".EstadoMesas[#Mesa].Rearme_CBx)) AND #ok_tension;
END_REGION

REGION Network 25: #PRV_Carga_OK_Inv
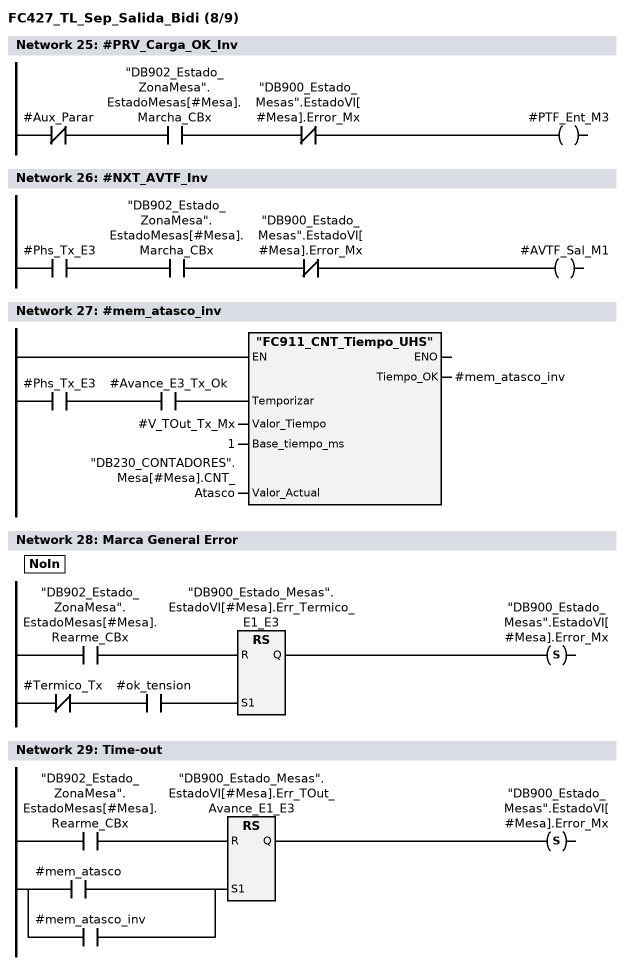
   RUNG wire#powerrail
      I_Contact( #Aux_Parar )
      Contact( "DB902_Estado_ZonaMesa".EstadoMesas[#Mesa].Marcha_CBx )
      I_Contact( "DB900_Estado_Mesas".EstadoVI[#Mesa].Error_Mx )
      Coil( #PTF_Ent_M3 )
   END_RUNG
   // the same network as SCL:
   #PTF_Ent_M3 := NOT #Aux_Parar AND "DB902_Estado_ZonaMesa".EstadoMesas[#Mesa].Marcha_CBx AND NOT "DB900_Estado_Mesas".EstadoVI[#Mesa].Error_Mx;
END_REGION

REGION Network 26: #NXT_AVTF_Inv
   RUNG wire#powerrail
      Contact( #Phs_Tx_E3 )
      Contact( "DB902_Estado_ZonaMesa".EstadoMesas[#Mesa].Marcha_CBx )
      I_Contact( "DB900_Estado_Mesas".EstadoVI[#Mesa].Error_Mx )
      Coil( #AVTF_Sal_M1 )
   END_RUNG
   // the same network as SCL:
   #AVTF_Sal_M1 := #Phs_Tx_E3 AND "DB902_Estado_ZonaMesa".EstadoMesas[#Mesa].Marcha_CBx AND NOT "DB900_Estado_Mesas".EstadoVI[#Mesa].Error_Mx;
END_REGION

REGION Network 27: #mem_atasco_inv
   RUNG wire#powerrail
      "FC911_CNT_Tiempo_UHS"(Temporizar := wire#w1, Valor_Tiempo := #V_TOut_Tx_Mx, Base_tiempo_ms := 1, Valor_Actual := "DB230_CONTADORES".Mesa[#Mesa].CNT_Atasco, Tiempo_OK => #mem_atasco_inv)
   END_RUNG
   RUNG wire#powerrail
      Contact( #Phs_Tx_E3 )
      Contact( #Avance_E3_Tx_Ok )
   END_RUNG wire#w1
   // the same network as SCL:
   "FC911_CNT_Tiempo_UHS"(Temporizar := #Phs_Tx_E3 AND #Avance_E3_Tx_Ok,
                          Valor_Tiempo := #V_TOut_Tx_Mx,
                          Base_tiempo_ms := 1,
                          Valor_Actual := "DB230_CONTADORES".Mesa[#Mesa].CNT_Atasco,
                          Tiempo_OK => #mem_atasco_inv);
END_REGION

REGION Network 28: Marca General Error
   Label( NoIn )
   RUNG wire#powerrail
      Contact( "DB902_Estado_ZonaMesa".EstadoMesas[#Mesa].Rearme_CBx )
      S_RS(operand := "DB900_Estado_Mesas".EstadoVI[#Mesa].Err_Termico_E1_E3, s1 := wire#w1)
      S_Coil( "DB900_Estado_Mesas".EstadoVI[#Mesa].Error_Mx )
   END_RUNG
   RUNG wire#powerrail
      I_Contact( #Termico_Tx )
      Contact( #ok_tension )
   END_RUNG wire#w1
   // the same network as SCL:
   NoIn:
   IF "DB902_Estado_ZonaMesa".EstadoMesas[#Mesa].Rearme_CBx THEN
       "DB900_Estado_Mesas".EstadoVI[#Mesa].Err_Termico_E1_E3 := FALSE;   // RS flip-flop
   END_IF;
   IF NOT #Termico_Tx AND #ok_tension THEN
       "DB900_Estado_Mesas".EstadoVI[#Mesa].Err_Termico_E1_E3 := TRUE;
   END_IF;
   IF "DB900_Estado_Mesas".EstadoVI[#Mesa].Err_Termico_E1_E3 THEN
       "DB900_Estado_Mesas".EstadoVI[#Mesa].Error_Mx := TRUE;
   END_IF;
END_REGION

REGION Network 29: Time-out
   RUNG wire#powerrail
      Contact( "DB902_Estado_ZonaMesa".EstadoMesas[#Mesa].Rearme_CBx )
      S_RS(operand := "DB900_Estado_Mesas".EstadoVI[#Mesa].Err_TOut_Avance_E1_E3, s1 := wire#w1)
      S_Coil( "DB900_Estado_Mesas".EstadoVI[#Mesa].Error_Mx )
   END_RUNG
   RUNG wire#powerrail
      Contact( #mem_atasco )
   END_RUNG wire#w1
   RUNG wire#powerrail
      Contact( #mem_atasco_inv )
   END_RUNG wire#w1
   // the same network as SCL:
   IF "DB902_Estado_ZonaMesa".EstadoMesas[#Mesa].Rearme_CBx THEN
       "DB900_Estado_Mesas".EstadoVI[#Mesa].Err_TOut_Avance_E1_E3 := FALSE;   // RS flip-flop
   END_IF;
   IF #mem_atasco OR #mem_atasco_inv THEN
       "DB900_Estado_Mesas".EstadoVI[#Mesa].Err_TOut_Avance_E1_E3 := TRUE;
   END_IF;
   IF "DB900_Estado_Mesas".EstadoVI[#Mesa].Err_TOut_Avance_E1_E3 THEN
       "DB900_Estado_Mesas".EstadoVI[#Mesa].Error_Mx := TRUE;
   END_IF;
END_REGION

REGION Network 30: Entradas Mesas
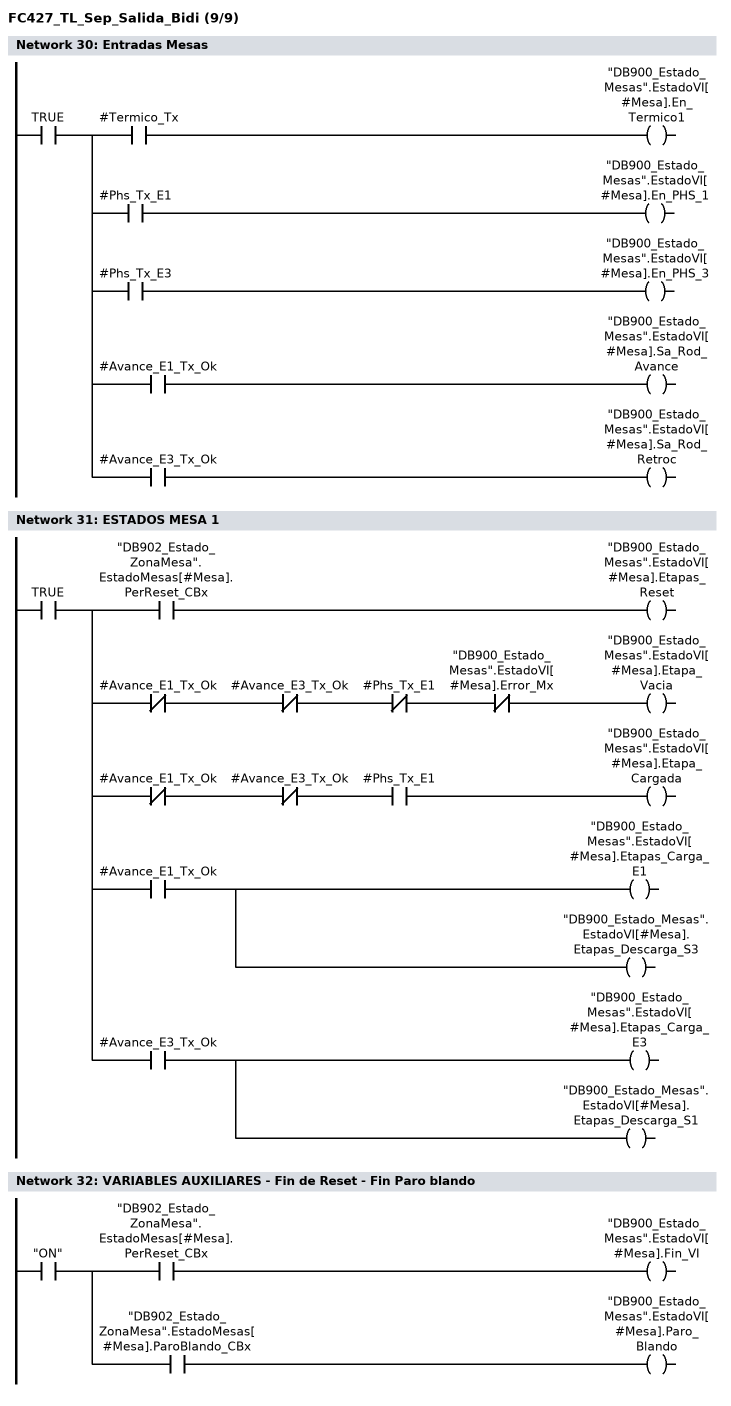
   RUNG wire#powerrail
      Contact( TRUE )
      wire#w1
      Contact( #Termico_Tx )
      Coil( "DB900_Estado_Mesas".EstadoVI[#Mesa].En_Termico1 )
   END_RUNG
   RUNG wire#w1
      Contact( #Phs_Tx_E1 )
      Coil( "DB900_Estado_Mesas".EstadoVI[#Mesa].En_PHS_1 )
   END_RUNG
   RUNG wire#w1
      Contact( #Phs_Tx_E3 )
      Coil( "DB900_Estado_Mesas".EstadoVI[#Mesa].En_PHS_3 )
   END_RUNG
   RUNG wire#w1
      Contact( #Avance_E1_Tx_Ok )
      Coil( "DB900_Estado_Mesas".EstadoVI[#Mesa].Sa_Rod_Avance )
   END_RUNG
   RUNG wire#w1
      Contact( #Avance_E3_Tx_Ok )
      Coil( "DB900_Estado_Mesas".EstadoVI[#Mesa].Sa_Rod_Retroc )
   END_RUNG
   // the same network as SCL:
   "DB900_Estado_Mesas".EstadoVI[#Mesa].En_Termico1 := TRUE AND #Termico_Tx;
   "DB900_Estado_Mesas".EstadoVI[#Mesa].En_PHS_1 := TRUE AND #Phs_Tx_E1;
   "DB900_Estado_Mesas".EstadoVI[#Mesa].En_PHS_3 := TRUE AND #Phs_Tx_E3;
   "DB900_Estado_Mesas".EstadoVI[#Mesa].Sa_Rod_Avance := TRUE AND #Avance_E1_Tx_Ok;
   "DB900_Estado_Mesas".EstadoVI[#Mesa].Sa_Rod_Retroc := TRUE AND #Avance_E3_Tx_Ok;
END_REGION

REGION Network 31: ESTADOS MESA 1
   RUNG wire#powerrail
      Contact( TRUE )
      wire#w1
      Contact( "DB902_Estado_ZonaMesa".EstadoMesas[#Mesa].PerReset_CBx )
      Coil( "DB900_Estado_Mesas".EstadoVI[#Mesa].Etapas_Reset )
   END_RUNG
   RUNG wire#w1
      I_Contact( #Avance_E1_Tx_Ok )
      I_Contact( #Avance_E3_Tx_Ok )
      I_Contact( #Phs_Tx_E1 )
      I_Contact( "DB900_Estado_Mesas".EstadoVI[#Mesa].Error_Mx )
      Coil( "DB900_Estado_Mesas".EstadoVI[#Mesa].Etapa_Vacia )
   END_RUNG
   RUNG wire#w1
      I_Contact( #Avance_E1_Tx_Ok )
      I_Contact( #Avance_E3_Tx_Ok )
      Contact( #Phs_Tx_E1 )
      Coil( "DB900_Estado_Mesas".EstadoVI[#Mesa].Etapa_Cargada )
   END_RUNG
   RUNG wire#w1
      Contact( #Avance_E1_Tx_Ok )
      wire#w2
      Coil( "DB900_Estado_Mesas".EstadoVI[#Mesa].Etapas_Carga_E1 )
   END_RUNG
   RUNG wire#w2
      Coil( "DB900_Estado_Mesas".EstadoVI[#Mesa].Etapas_Descarga_S3 )
   END_RUNG
   RUNG wire#w1
      Contact( #Avance_E3_Tx_Ok )
      wire#w3
      Coil( "DB900_Estado_Mesas".EstadoVI[#Mesa].Etapas_Carga_E3 )
   END_RUNG
   RUNG wire#w3
      Coil( "DB900_Estado_Mesas".EstadoVI[#Mesa].Etapas_Descarga_S1 )
   END_RUNG
   // the same network as SCL:
   "DB900_Estado_Mesas".EstadoVI[#Mesa].Etapas_Reset := TRUE AND "DB902_Estado_ZonaMesa".EstadoMesas[#Mesa].PerReset_CBx;
   "DB900_Estado_Mesas".EstadoVI[#Mesa].Etapa_Vacia := TRUE AND NOT #Avance_E1_Tx_Ok AND NOT #Avance_E3_Tx_Ok AND NOT #Phs_Tx_E1 AND NOT "DB900_Estado_Mesas".EstadoVI[#Mesa].Error_Mx;
   "DB900_Estado_Mesas".EstadoVI[#Mesa].Etapa_Cargada := TRUE AND NOT #Avance_E1_Tx_Ok AND NOT #Avance_E3_Tx_Ok AND #Phs_Tx_E1;
   "DB900_Estado_Mesas".EstadoVI[#Mesa].Etapas_Carga_E1 := TRUE AND #Avance_E1_Tx_Ok;
   "DB900_Estado_Mesas".EstadoVI[#Mesa].Etapas_Descarga_S3 := TRUE AND #Avance_E1_Tx_Ok;
   "DB900_Estado_Mesas".EstadoVI[#Mesa].Etapas_Carga_E3 := TRUE AND #Avance_E3_Tx_Ok;
   "DB900_Estado_Mesas".EstadoVI[#Mesa].Etapas_Descarga_S1 := TRUE AND #Avance_E3_Tx_Ok;
END_REGION

REGION Network 32: VARIABLES AUXILIARES - Fin de Reset - Fin Paro blando
   RUNG wire#powerrail
      Contact( "ON" )
      wire#w1
      Contact( "DB902_Estado_ZonaMesa".EstadoMesas[#Mesa].PerReset_CBx )
      Coil( "DB900_Estado_Mesas".EstadoVI[#Mesa].Fin_VI )
   END_RUNG
   RUNG wire#w1
      Contact( "DB902_Estado_ZonaMesa".EstadoMesas[#Mesa].ParoBlando_CBx )
      Coil( "DB900_Estado_Mesas".EstadoVI[#Mesa].Paro_Blando )
   END_RUNG
   // the same network as SCL:
   "DB900_Estado_Mesas".EstadoVI[#Mesa].Fin_VI := "ON" AND "DB902_Estado_ZonaMesa".EstadoMesas[#Mesa].PerReset_CBx;
   "DB900_Estado_Mesas".EstadoVI[#Mesa].Paro_Blando := "ON" AND "DB902_Estado_ZonaMesa".EstadoMesas[#Mesa].ParoBlando_CBx;
END_REGION
END_FUNCTION
